// TIA Portal V18 export
TYPE "TM_Count_Man_Out"
   STRUCT
      SLOT_0 : Real;
      SLOT_1 : Real;
      LD_SLOT_0_1 : Byte;
      SW_GATE : Bool;
      TM_CTRL_DQ0 : Bool;
      TM_CTRL_DQ1 : Bool;
      SET_DQ0 : Bool;
      SET_DQ1 : Bool;
      EN_SYNC_UP : Bool;
      EN_SYNC_DN : Bool;
      EN_CAPTURE : Bool;
      RES_ERROR : Bool;
      RES_EVENT : Bool;
      Reserved1 : Bool;
      Reserved2 : Bool;
      Reserved3 : Bool;
      Reserved4 : Bool;
      Reserved5 : Bool;
      SET_DIR : Bool;
      Reserved : Byte;
   END_STRUCT;
END_TYPE
